(* CODESYS project codesys-poc

Project tree, tasks and I/O mapping:
  CODESYS_Control_RTE_V3 : CODESYS Control RTE V3, CODESYS, order no. 305017, version 3.5.21.10
    application Application
  Device : CODESYS Control Win V3 x64, CODESYS, version 3.5.21.10
    application Application
      libraries: Standard, 3.5.18.0 (System); Test Manager IEC Unit Test, 5.1.0.0 (Intern)
      task MainTask (cyclic, interval t#20ms, priority 1) calls PLC_PRG
      task VISU_TASK (cyclic, interval 100 ms, priority 31) calls VisuElems.Visu_Prg
      Antenna/
        function block Antenna [ST]: DiscesaAnteriore, DiscesaAnterioreEnabled, DiscesaAnterioreStop
        interface IAntenna: DiscesaAnteriore, DiscesaAnterioreEnabled, DiscesaAnterioreStop
        function block ManagerAntenna [ST]
      ArganoPrincipale/
        function block Argano [ST]: Arrotola
        interface IArgano: Arrotola
        function block ManagerArgano [ST]
      Controls/
        Joystyck/
          function block Joystick2 [CFC]
          function block Joystick3 [SFC]
          function block Joystick4 [FBD]
          function block Joystick [ST]
      Motore/
        interface IMotore: Accendi, GiriMotore, SpegniMotore
        function block MotoreDiesel [CFC]: Accendi, GiriMotore
      program PLC_PRG [ST]
      Rotary/
        interface IRotary: ClickClick, Rotate, RotateStop, SetCilindrata, SpinOff
        function block ManagerRotary [ST]
        function block Rotary [ST]: ClickClick, Rotate, RotateStop, SetCilindrata, SpinOff
        function block TestRotation_1 [ST]: Abort, Execute, Setup, Teardown
        function block TestRotation [ST]: Abort, Execute, Setup, Teardown
      Valvole/
        function block DistributoreValvole [ST]: openV1, openV2
        interface IDistributoreValvole: openV1, openV2
        interface IPompa: Portata
        function block Pompa [ST]: Portata
      visualisation Visualization_1
    application Application
      libraries: Standard, 3.5.18.0 (System)
      task MainTask (cyclic, interval t#20ms, priority 1) calls PLC_PRG
      task VISU_TASK (cyclic, interval 100 ms, priority 31) calls VisuElems.Visu_Prg
      Antenna/
        function block Antenna [ST]: DiscesaAnteriore, DiscesaAnterioreEnabled, DiscesaAnterioreStop
        interface IAntenna: DiscesaAnteriore, DiscesaAnterioreEnabled, DiscesaAnterioreStop
        function block ManagerAntenna [ST]
      ArganoPrincipale/
        function block Argano [ST]: Arrotola
        interface IArgano: Arrotola
        function block ManagerArgano [ST]
      Controls/
        Joystyck/
          function block Joystick2 [CFC]
          function block Joystick3 [SFC]
          function block Joystick4 [FBD]
          function block Joystick [ST]
      program PLC_PRG [ST]
      Rotary/
        interface IRotary: ClickClick, Rotate, RotateStop, SetCilindrata, SpinOff
        function block ManagerRotary [ST]
        function block Rotary [ST]: ClickClick, Rotate, RotateStop, SetCilindrata, SpinOff
      Valvole/
        function block DistributoreValvole [ST]: openV1, openV2
        interface IDistributoreValvole: openV1, openV2
        interface IPompa: Portata
        function block Pompa [ST]: Portata
      visualisation Visualization_1
    application Application
      libraries: Standard, 3.5.18.0 (System); Test Manager IEC Unit Test, 5.1.0.0 (Intern)
      task MainTask (cyclic, interval t#20ms, priority 1) calls PLC_PRG
      task VISU_TASK (cyclic, interval 100 ms, priority 31) calls VisuElems.Visu_Prg
      Antenna/
        function block Antenna [ST]: DiscesaAnteriore, DiscesaAnterioreEnabled, DiscesaAnterioreStop
        interface IAntenna: DiscesaAnteriore, DiscesaAnterioreEnabled, DiscesaAnterioreStop
        function block ManagerAntenna [ST]
      ArganoPrincipale/
        function block Argano [ST]: Arrotola
        interface IArgano: Arrotola
        function block ManagerArgano [ST]
      Controls/
        Joystyck/
          ClassDiagram_Control
          interface IJoystick: axisX, axisY, enabled, triggered
          function block Joystick2 [CFC]
          function block Joystick3 [SFC]
          function block Joystick4 [FBD]: axisX, axisY, enabled, safe, triggered
          function block Joystick [ST]: axisX, axisY, enabled, safe, triggered
      interface ISafeManaged: safe
      Motore/
        interface IMotore: Accendi, GiriMotore, SpegniMotore
        function block MotoreDiesel [CFC]: Accendi, GiriMotore
      program PLC_PRG [ST]
      Rotary/
        function block AutoRotate [CFC]: direction, enabled, speed
        ClassDiagram
        interface IAutoRotate: direction, enabled, speed
        interface IRotary: ClickClick, Rotate, RotateStop, SetCilindrata, SpinOff
        function block ManagerRotary [ST]
        function block Rotary [ST]: ClickClick, Rotate, RotateStop, safe, SetCilindrata, SpinOff
        function block TestRotation_1 [ST]: Abort, Execute, Setup, Teardown
        function block TestRotation [ST]: Abort, Execute, Setup, Teardown
      Valvole/
        function block DistributionValve [ST]: GetActual, GetTarget, Open, safe, openV2
        interface IDistributionValve: GetActual, GetTarget, Open, openV2
        interface IPompa: Portata
        function block Pompa [ST]: Portata
      visualisation Visualization_1
  Generated Unit Tests/
  text list GlobalTextList
*)

// Device/Application/PLC_PRG
PROGRAM PLC_PRG
VAR
	joystick1 : Joystick;
    joystick : Joystick4;
	
    rotary : Rotary;
	managerRotary: ManagerRotary;
	
	antenna: Antenna;
	managerAntenna: ManagerAntenna;
	
	argano: Argano;
	managerArgano: ManagerArgano;
	
	pompa : Pompa;
	distributore: DistributoreValvole;
	
	safe : BOOL;
	// Generated by IEC Unit Test
	xDone: BOOL;
	// Generated by IEC Unit Test
	xError: BOOL;
	// Generated by IEC Unit Test
	instTESTCASE: TestRotation;
END_VAR

joystick1.Safe := safe;
joystick.Safe := safe;

distributore.pompa := pompa;

managerRotary.joystick := joystick1;
managerRotary.rotary := rotary;

managerAntenna.joystick := joystick;
managerAntenna.antenna := antenna;

managerArgano.argano := argano;
managerArgano.antenna := antenna;

rotary.Safe := safe;
rotary.distributore := distributore;

// controlli
joystick();
joystick1();

// gruppi
antenna();
argano();
pompa();
distributore();

// manager
managerRotary();
managerAntenna(); // managerAntenna(antenna := antenna, joystick := joystick);
managerArgano();

END_PROGRAM

// Device/Application/Controls/Joystyck/Joystick
FUNCTION_BLOCK Joystick
VAR_INPUT
	Safe: BOOL;
	Trigger: BOOL;
END_VAR
VAR_OUTPUT
	Enabled: BOOL;
	EnabledOR: BOOL;
END_VAR
VAR
	EnabledInner: BOOL;
END_VAR

Enabled := Safe AND Trigger;
EnabledOR := Safe OR Trigger;

END_FUNCTION_BLOCK

// Device/Application/Controls/Joystyck/Joystick
FUNCTION_BLOCK Joystick
VAR_INPUT
	Safe: BOOL;
	Trigger: BOOL;
END_VAR
VAR_OUTPUT
	Enabled: BOOL;
	EnabledOR: BOOL;
END_VAR
VAR
	EnabledInner: BOOL;
END_VAR

Enabled := Safe AND Trigger;
EnabledOR := Safe OR Trigger;

END_FUNCTION_BLOCK

// Device/Application/Controls/Joystyck/Joystick
FUNCTION_BLOCK Joystick
VAR_INPUT
	Safe: BOOL;
	Trigger: BOOL;
END_VAR
VAR_OUTPUT
	Enabled: BOOL;
	EnabledOR: BOOL;
END_VAR
VAR
	EnabledInner: BOOL;
END_VAR

Enabled := Safe AND Trigger;
EnabledOR := Safe OR Trigger;

{warning 'Aggiungi implementazione della proprietà'}
PROPERTY axisX : REAL
GET
END_GET
END_PROPERTY

{warning 'Aggiungi implementazione della proprietà'}
PROPERTY axisY : REAL
GET
axisY := 0.0;
END_GET
END_PROPERTY

{warning 'Aggiungi implementazione della proprietà'}
PROPERTY enabled : BOOL
GET
END_GET
END_PROPERTY

{warning 'Aggiungi implementazione della proprietà'}
PROPERTY safe : BOOL
GET
safe := _safe;
END_GET
END_PROPERTY

{warning 'Aggiungi implementazione della proprietà'}
PROPERTY triggered : BOOL
GET
END_GET
END_PROPERTY

END_FUNCTION_BLOCK

// Device/Application/Valvole/Pompa
FUNCTION_BLOCK Pompa IMPLEMENTS IPompa
VAR_INPUT
	_portata: REAL;
END_VAR
VAR_OUTPUT
END_VAR
VAR
END_VAR

PROPERTY Portata : REAL
GET
Portata := _portata;
END_GET
SET
_portata := Portata;
END_SET
END_PROPERTY

END_FUNCTION_BLOCK

// Device/Application/Valvole/Pompa
FUNCTION_BLOCK Pompa IMPLEMENTS IPompa
VAR_INPUT
	_portata: REAL;
END_VAR
VAR_OUTPUT
END_VAR
VAR
END_VAR

PROPERTY Portata : REAL
GET
Portata := _portata;
END_GET
SET
_portata := Portata;
END_SET
END_PROPERTY

END_FUNCTION_BLOCK

// Device/Application/Valvole/Pompa
FUNCTION_BLOCK Pompa IMPLEMENTS IPompa
VAR_INPUT
	_portata: REAL;
END_VAR
VAR_OUTPUT
END_VAR
VAR
END_VAR

PROPERTY Portata : REAL
GET
Portata := _portata;
END_GET
SET
_portata := Portata;
END_SET
END_PROPERTY

END_FUNCTION_BLOCK

// Device/Application/Valvole/IPompa
INTERFACE IPompa

PROPERTY Portata : REAL
GET
END_GET
SET
END_SET
END_PROPERTY

END_INTERFACE

// Device/Application/Valvole/IPompa
INTERFACE IPompa

PROPERTY Portata : REAL
GET
END_GET
SET
END_SET
END_PROPERTY

END_INTERFACE

// Device/Application/Valvole/IPompa
INTERFACE IPompa

PROPERTY Portata : REAL
GET
END_GET
SET
END_SET
END_PROPERTY

END_INTERFACE

// Device/Application/Rotary/ManagerRotary
FUNCTION_BLOCK ManagerRotary
VAR_INPUT
	rotary: IRotary;
	joystick: Joystick;
END_VAR
VAR_OUTPUT
END_VAR
VAR
	rotationEnabled: BOOL;
END_VAR

// rotary.rotate = joystick.Enabled;
rotationEnabled := joystick.Enabled;

// SOL 1
IF rotationEnabled THEN
	rotary.Rotate(Side := 'LEFT', Speed := 10);
	// rampa(actual, desired);
ELSE
	rotary.RotateStop();
	// rotary.Rotate(Side := 'null', Speed := 0);
	// rampa(actual, 0);
END_IF

// SOL 2
//
// ManagerRotary:
//
// rotary.Rotate(rotationEnabled, Side := 'LEFT', Speed := 10);
//
// Rotary:
//
// IF rotationEnabled THEN
// 	  Rotate(rotationEnabled, Side := 'LEFT', Speed := 10);
// ELSE
// 	  Rotate(rotationEnabled, Side := 'LEFT', Speed := 0);
// END_IF


// SOL 3
//
// rotary.RotateStop(); SOLO SE FARE LO STOP E' IDEMPOTENTE
// IF rotationEnabled THEN
// 	rotary.Rotate(Side := 'LEFT', Speed := 10);
// END_IF

END_FUNCTION_BLOCK

// Device/Application/Rotary/Rotary
FUNCTION_BLOCK Rotary IMPLEMENTS IRotary
VAR_INPUT
	Safe: BOOL;
	distributore: IDistributoreValvole;
END_VAR
VAR_OUTPUT
END_VAR
VAR
    InvocationCount : INT := 0; // Counter for total method invocations
END_VAR

METHOD ClickClick
VAR
    clicked : BOOL;
END_VAR
// Simulate click-click behavior
clicked := TRUE; // Placeholder for actual logic

// IF Safe THEN
// 	InvocationCount := InvocationCount + 1; // Increase method call count
// END_IF;
END_METHOD

METHOD Rotate
VAR_INPUT
    Side : STRING;  // "Left" or "Right"
    Speed : REAL;   // Rotation speed
END_VAR
VAR_OUTPUT
	ActualSpeed: REAL;
END_VAR
// Simulated behavior
// direction := TO_UPPER(Side);
IF Side = 'LEFT' THEN
    // Do something for left rotation
    // For demo, just print or simulate log
    ; // Can add logging or effect
ELSIF Side = 'RIGHT' THEN
    // Do something for right rotation
    ;
ELSE
    ; // Invalid direction
END_IF;

InvocationCount := InvocationCount + 1; // Increase method call count
distributore.openV1(Speed);
ActualSpeed := Speed;
END_METHOD

METHOD RotateStop
distributore.openV1(0.0);
END_METHOD

METHOD SetCilindrata
// IF Safe THEN
// 	InvocationCount := InvocationCount + 1; // Increase method call count
// END_IF;
END_METHOD

METHOD SpinOff
VAR_INPUT
    dummy : BOOL;
END_VAR
// Simulate spinoff behavior
// For example: Do something when spinning off

// IF Safe THEN
// 	InvocationCount := InvocationCount + 1; // Increase method call count
// END_IF;
END_METHOD

END_FUNCTION_BLOCK

// Device/Application/Rotary/Rotary
FUNCTION_BLOCK Rotary IMPLEMENTS IRotary
VAR_INPUT
	Safe: BOOL;
	distributore: IDistributoreValvole;
END_VAR
VAR_OUTPUT
END_VAR
VAR
    InvocationCount : INT := 0; // Counter for total method invocations
END_VAR

METHOD ClickClick
VAR
    clicked : BOOL;
END_VAR
// Simulate click-click behavior
clicked := TRUE; // Placeholder for actual logic

// IF Safe THEN
// 	InvocationCount := InvocationCount + 1; // Increase method call count
// END_IF;
END_METHOD

METHOD Rotate
VAR_INPUT
    Side : STRING;  // "Left" or "Right"
    Speed : REAL;   // Rotation speed
END_VAR
VAR
    direction : STRING;
END_VAR
// Simulated behavior
// direction := TO_UPPER(Side);
IF Side = 'LEFT' THEN
    // Do something for left rotation
    // For demo, just print or simulate log
    ; // Can add logging or effect
ELSIF Side = 'RIGHT' THEN
    // Do something for right rotation
    ;
ELSE
    ; // Invalid direction
END_IF;

InvocationCount := InvocationCount + 1; // Increase method call count
distributore.openV1(10.0);
END_METHOD

METHOD RotateStop
distributore.openV1(0.0);
END_METHOD

METHOD SetCilindrata
// IF Safe THEN
// 	InvocationCount := InvocationCount + 1; // Increase method call count
// END_IF;
END_METHOD

METHOD SpinOff
VAR_INPUT
    dummy : BOOL;
END_VAR
// Simulate spinoff behavior
// For example: Do something when spinning off

// IF Safe THEN
// 	InvocationCount := InvocationCount + 1; // Increase method call count
// END_IF;
END_METHOD

END_FUNCTION_BLOCK

// Device/Application/Rotary/Rotary
FUNCTION_BLOCK Rotary IMPLEMENTS IRotary, ISafeManaged
VAR_INPUT
	distributore: IDistributionValve;
END_VAR
VAR_OUTPUT
END_VAR
VAR
    _safe: BOOL;
	invocationCount : INT := 0; // Counter for total method invocations
END_VAR

METHOD ClickClick
VAR
    clicked : BOOL;
END_VAR
// Simulate click-click behavior
clicked := TRUE; // Placeholder for actual logic

// IF Safe THEN
// 	InvocationCount := InvocationCount + 1; // Increase method call count
// END_IF;
END_METHOD

METHOD Rotate
VAR_INPUT
    side : STRING;  // "Left" or "Right"
    speed : REAL;   // Rotation speed
END_VAR
VAR_OUTPUT
	actualSpeed: REAL;
END_VAR
// Simulated behavior
// direction := TO_UPPER(Side);
IF Side = 'LEFT' THEN
    // Do something for left rotation
    // For demo, just print or simulate log
    ; // Can add logging or effect
ELSIF Side = 'RIGHT' THEN
    // Do something for right rotation
    ;
ELSE
    ; // Invalid direction
END_IF;

invocationCount := invocationCount + 1; // Increase method call count
distributionValve.Open(1, Speed);
actualSpeed := speed;
END_METHOD

METHOD RotateStop
distributionValve.open(1, 0.0);
END_METHOD

{warning 'Aggiungi implementazione della proprietà'}
PROPERTY safe : BOOL
GET
safe := _safe;
END_GET
END_PROPERTY

METHOD SetCilindrata
// IF Safe THEN
// 	InvocationCount := InvocationCount + 1; // Increase method call count
// END_IF;
END_METHOD

METHOD SpinOff
VAR_INPUT
    dummy : BOOL;
END_VAR
// Simulate spinoff behavior
// For example: Do something when spinning off

// IF Safe THEN
// 	InvocationCount := InvocationCount + 1; // Increase method call count
// END_IF;
END_METHOD

END_FUNCTION_BLOCK

// Device/Application/Rotary/IRotary
INTERFACE IRotary

METHOD ClickClick
VAR_INPUT
END_VAR
END_METHOD

METHOD Rotate
VAR_INPUT
    Side : STRING;  // "Left" or "Right"
    Speed : REAL;   // Rotation speed
END_VAR
VAR_OUTPUT
	ActualSpeed: REAL;
END_VAR
END_METHOD

METHOD RotateStop
VAR_INPUT
END_VAR
END_METHOD

METHOD SetCilindrata
VAR_INPUT
END_VAR
END_METHOD

METHOD SpinOff
VAR_INPUT
    dummy : BOOL;
END_VAR
END_METHOD

END_INTERFACE

// Device/Application/Rotary/IRotary
INTERFACE IRotary

METHOD ClickClick
VAR_INPUT
END_VAR
END_METHOD

METHOD Rotate
VAR_INPUT
    Side : STRING;  // "Left" or "Right"
    Speed : REAL;   // Rotation speed
END_VAR
END_METHOD

METHOD RotateStop
VAR_INPUT
END_VAR
END_METHOD

METHOD SetCilindrata
VAR_INPUT
END_VAR
END_METHOD

METHOD SpinOff
VAR_INPUT
    dummy : BOOL;
END_VAR
END_METHOD

END_INTERFACE

// Device/Application/Rotary/IRotary
INTERFACE IRotary

METHOD ClickClick
VAR_INPUT
END_VAR
END_METHOD

METHOD Rotate
VAR_INPUT
    Side : STRING;  // "Left" or "Right"
    Speed : REAL;   // Rotation speed
END_VAR
VAR_OUTPUT
	ActualSpeed: REAL;
END_VAR
END_METHOD

METHOD RotateStop
VAR_INPUT
END_VAR
END_METHOD

METHOD SetCilindrata
VAR_INPUT
END_VAR
END_METHOD

METHOD SpinOff
END_METHOD

END_INTERFACE

// Device/Application/ISafeManaged
INTERFACE ISafeManaged

PROPERTY safe : BOOL
GET
END_GET
END_PROPERTY

END_INTERFACE

// Device/Application/Valvole/IDistributionValve
INTERFACE IDistributionValve

METHOD GetActual : REAL
VAR_INPUT
	idValve: INT;
END_VAR
END_METHOD

METHOD GetTarget : REAL
VAR_INPUT
	idValve : INT;
END_VAR
END_METHOD

METHOD Open
VAR_INPUT
	idValve: INT;
	flow: REAL;
END_VAR
END_METHOD

METHOD openV2
VAR_INPUT
	portata: REAL;
END_VAR
END_METHOD

END_INTERFACE

// Device/Application/Valvole/DistributionValve
FUNCTION_BLOCK DistributionValve IMPLEMENTS IDistributionValve, ISafeManaged
VAR_INPUT
	pump : IPump;
END_VAR
VAR_OUTPUT
END_VAR
VAR
	_vActual: ARRAY[1..10] OF REAL := [0, 0, 0, 0, 0, 0, 0, 0, 0, 0];
	_vTarget: ARRAY[1..10] OF REAL := [0, 0, 0, 0, 0, 0, 0, 0, 0, 0];
	flowSum : REAL := 0.0; // Reset flow accumulator
	firstValve: INT := -1;
	i: INT := 1;
	count: INT := 0;
END_VAR

flowSum := 0.0; // Reset flow accumulator

FOR i := 1 TO 10 DO
    IF _vTarget[i] <> 0 THEN
		flowSum := flowSum + _vActual[i];        
		count := count + 1;
		_vActual[i] := _vTarget[i];
		firstValve := i;
    ELSE
        _vActual[i] := 0.0;
    END_IF
END_FOR

IF count = 1 THEN
	pump.flow := _vActual[firstValve];	
	_vActual[firstValve] := 100.0;
ELSE 
	pump.flow := flowSum;
END_IF

METHOD GetActual : REAL
VAR_INPUT
	idValve	: INT;
END_VAR
getActual := _vActual[idValve];
END_METHOD

METHOD GetTarget : REAL
VAR_INPUT
	idValve : INT;
END_VAR
getTarget := _vTarget[idValve];
END_METHOD

METHOD Open
VAR_INPUT
	idValve: INT;	
	flow: REAL;
END_VAR
_vTarget[idValve] := flow;
END_METHOD

{warning 'Aggiungi implementazione della proprietà'}
PROPERTY safe : BOOL
GET
END_GET
END_PROPERTY

METHOD openV2
VAR_INPUT
	portata: REAL;
END_VAR
_v2 := portata;
END_METHOD

END_FUNCTION_BLOCK

// Device/Application/Valvole/IDistributoreValvole
INTERFACE IDistributoreValvole

METHOD openV1
VAR_INPUT
	portata: REAL;
END_VAR
END_METHOD

METHOD openV2
VAR_INPUT
	portata: REAL;
END_VAR
END_METHOD

END_INTERFACE

// Device/Application/Valvole/IDistributoreValvole
INTERFACE IDistributoreValvole

METHOD openV1
VAR_INPUT
	portata: REAL;
END_VAR
END_METHOD

METHOD openV2
VAR_INPUT
	portata: REAL;
END_VAR
END_METHOD

END_INTERFACE

// Device/Application/Rotary/ManagerRotary
FUNCTION_BLOCK ManagerRotary
VAR_INPUT
	rotary: IRotary;
	joystick: Joystick;
END_VAR
VAR_OUTPUT
END_VAR
VAR
	rotationEnabled: BOOL;
END_VAR

// rotary.rotate = joystick.Enabled;
rotationEnabled := joystick.Enabled;

// SOL 1
IF rotationEnabled THEN
	rotary.Rotate(Side := 'LEFT', Speed := 10);
	// rampa(actual, desired);
ELSE
	// rotary.RotateStop();
	rotary.Rotate(Side := 'null', Speed := 0);
	// rampa(actual, 0);
END_IF

// SOL 2
//
// ManagerRotary:
//
// rotary.Rotate(rotationEnabled, Side := 'LEFT', Speed := 10);
//
// Rotary:
//
// IF rotationEnabled THEN
// 	  Rotate(rotationEnabled, Side := 'LEFT', Speed := 10);
// ELSE
// 	  Rotate(rotationEnabled, Side := 'LEFT', Speed := 0);
// END_IF


// SOL 3
//
// rotary.RotateStop(); SOLO SE FARE LO STOP E' IDEMPOTENTE
// IF rotationEnabled THEN
// 	rotary.Rotate(Side := 'LEFT', Speed := 10);
// END_IF

END_FUNCTION_BLOCK

// Device/Application/Rotary/ManagerRotary
FUNCTION_BLOCK ManagerRotary
VAR_INPUT
	rotary: IRotary;
	joystick: IJoystick;
END_VAR
VAR_OUTPUT
END_VAR
VAR
	_rotationEnabled: BOOL;
END_VAR

// rotary.rotate = joystick.Enabled;
_rotationEnabled := joystick.Enabled;

// SOL 1
IF _rotationEnabled THEN
	rotary.Rotate(Side := 'LEFT', Speed := 10);
	// rampa(actual, desired);
ELSE
	rotary.RotateStop();
	// rotary.Rotate(Side := 'null', Speed := 0);
	// rampa(actual, 0);
END_IF

// SOL 2
//
// ManagerRotary:
//
// rotary.Rotate(rotationEnabled, Side := 'LEFT', Speed := 10);
//
// Rotary:
//
// IF rotationEnabled THEN
// 	  Rotate(rotationEnabled, Side := 'LEFT', Speed := 10);
// ELSE
// 	  Rotate(rotationEnabled, Side := 'LEFT', Speed := 0);
// END_IF


// SOL 3
//
// rotary.RotateStop(); SOLO SE FARE LO STOP E' IDEMPOTENTE
// IF rotationEnabled THEN
// 	rotary.Rotate(Side := 'LEFT', Speed := 10);
// END_IF

END_FUNCTION_BLOCK

// Device/Application/Controls/Joystyck/IJoystick
INTERFACE IJoystick EXTENDS ISafeManaged

PROPERTY axisX : REAL
GET
END_GET
END_PROPERTY

PROPERTY axisY : REAL
GET
END_GET
END_PROPERTY

PROPERTY enabled : BOOL
GET
END_GET
END_PROPERTY

PROPERTY triggered : BOOL
GET
END_GET
END_PROPERTY

END_INTERFACE

// Device/Application/Antenna/ManagerAntenna
FUNCTION_BLOCK ManagerAntenna
VAR_INPUT
	antenna: IAntenna;
	joystick: Joystick4;
END_VAR
VAR_OUTPUT
END_VAR
VAR
END_VAR

IF joystick.Enabled THEN
	antenna.DiscesaAnteriore();
ELSE
	antenna.DiscesaAnterioreStop();
END_IF

END_FUNCTION_BLOCK

// Device/Application/Antenna/Antenna
FUNCTION_BLOCK Antenna IMPLEMENTS IAntenna
VAR
	_discesaanterioreenabled : BOOL := FALSE; // Internal state
END_VAR

METHOD DiscesaAnteriore
_discesaanterioreenabled := TRUE;
END_METHOD

PROPERTY PUBLIC DiscesaAnterioreEnabled : BOOL
GET
DiscesaAnterioreEnabled := _discesaanterioreenabled;
END_GET
END_PROPERTY

METHOD DiscesaAnterioreStop
_discesaanterioreenabled := FALSE;
END_METHOD

END_FUNCTION_BLOCK

// Device/Application/Antenna/Antenna
FUNCTION_BLOCK Antenna IMPLEMENTS IAntenna
VAR
	_discesaanterioreenabled : BOOL := FALSE; // Internal state
END_VAR

METHOD DiscesaAnteriore
_discesaanterioreenabled := TRUE;
END_METHOD

PROPERTY PUBLIC DiscesaAnterioreEnabled : BOOL
GET
DiscesaAnterioreEnabled := _discesaanterioreenabled;
END_GET
END_PROPERTY

METHOD DiscesaAnterioreStop
_discesaanterioreenabled := FALSE;
END_METHOD

END_FUNCTION_BLOCK

// Device/Application/Antenna/Antenna
FUNCTION_BLOCK Antenna IMPLEMENTS IAntenna
VAR
	_discesaanterioreenabled : BOOL := FALSE; // Internal state
END_VAR

METHOD DiscesaAnteriore
_discesaanterioreenabled := TRUE;
END_METHOD

PROPERTY PUBLIC DiscesaAnterioreEnabled : BOOL
GET
DiscesaAnterioreEnabled := _discesaanterioreenabled;
END_GET
END_PROPERTY

METHOD DiscesaAnterioreStop
_discesaanterioreenabled := FALSE;
END_METHOD

END_FUNCTION_BLOCK

// Device/Application/Antenna/IAntenna
INTERFACE IAntenna

METHOD DiscesaAnteriore
VAR_INPUT
END_VAR
END_METHOD

PROPERTY PUBLIC DiscesaAnterioreEnabled : BOOL
GET
END_GET
END_PROPERTY

METHOD DiscesaAnterioreStop
VAR_INPUT
END_VAR
END_METHOD

END_INTERFACE

// Device/Application/Antenna/IAntenna
INTERFACE IAntenna

METHOD DiscesaAnteriore
VAR_INPUT
END_VAR
END_METHOD

PROPERTY PUBLIC DiscesaAnterioreEnabled : BOOL
GET
END_GET
END_PROPERTY

METHOD DiscesaAnterioreStop
VAR_INPUT
END_VAR
END_METHOD

END_INTERFACE

// Device/Application/Antenna/IAntenna
INTERFACE IAntenna

METHOD DiscesaAnteriore
VAR_INPUT
END_VAR
END_METHOD

PROPERTY PUBLIC DiscesaAnterioreEnabled : BOOL
GET
END_GET
END_PROPERTY

METHOD DiscesaAnterioreStop
VAR_INPUT
END_VAR
END_METHOD

END_INTERFACE

// Device/Application/Antenna/ManagerAntenna
FUNCTION_BLOCK ManagerAntenna
VAR_INPUT
	antenna: IAntenna;
	joystick: Joystick4;
END_VAR
VAR_OUTPUT
END_VAR
VAR
END_VAR

IF joystick.Enabled THEN
	antenna.DiscesaAnteriore();
ELSE
	antenna.DiscesaAnterioreStop();
END_IF

END_FUNCTION_BLOCK

// Device/Application/Antenna/ManagerAntenna
FUNCTION_BLOCK ManagerAntenna
VAR_INPUT
	antenna: IAntenna;
	joystick: Joystick4;
END_VAR
VAR_OUTPUT
END_VAR
VAR
END_VAR

IF joystick.Enabled THEN
	antenna.DiscesaAnteriore();
ELSE
	antenna.DiscesaAnterioreStop();
END_IF

END_FUNCTION_BLOCK

// Device/Application/Controls/Joystyck/Joystick4
FUNCTION_BLOCK Joystick4
VAR_INPUT
	Safe: BOOL;
END_VAR
VAR_OUTPUT
	Enabled: BOOL;
END_VAR
VAR
	Trigger: BOOL;
END_VAR

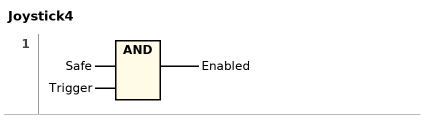
// NETWORK 1
Enabled := Safe AND Trigger;

END_FUNCTION_BLOCK

// Device/Application/Controls/Joystyck/Joystick4
FUNCTION_BLOCK Joystick4
VAR_INPUT
	Safe: BOOL;
END_VAR
VAR_OUTPUT
	Enabled: BOOL;
END_VAR
VAR
	Trigger: BOOL;
END_VAR

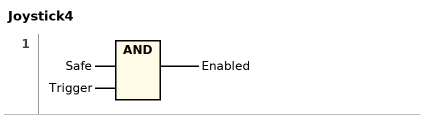
// NETWORK 1
Enabled := Safe AND Trigger;

END_FUNCTION_BLOCK

// Device/Application/Controls/Joystyck/Joystick4
FUNCTION_BLOCK Joystick4
VAR_INPUT
	Safe: BOOL;
END_VAR
VAR_OUTPUT
	Enabled: BOOL;
END_VAR
VAR
	Trigger: BOOL;
END_VAR

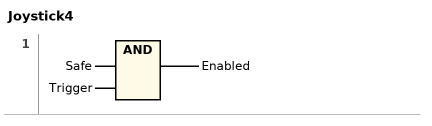
// NETWORK 1
Enabled := Safe AND Trigger;

{warning 'Aggiungi implementazione della proprietà'}
PROPERTY axisX : REAL
GET
END_GET
END_PROPERTY

{warning 'Aggiungi implementazione della proprietà'}
PROPERTY axisY : REAL
GET
END_GET
END_PROPERTY

{warning 'Aggiungi implementazione della proprietà'}
PROPERTY enabled : BOOL
GET
END_GET
END_PROPERTY

{warning 'Aggiungi implementazione della proprietà'}
PROPERTY safe : BOOL
GET
END_GET
END_PROPERTY

{warning 'Aggiungi implementazione della proprietà'}
PROPERTY triggered : BOOL
GET
END_GET
END_PROPERTY

END_FUNCTION_BLOCK

// Device/Application/ArganoPrincipale/ManagerArgano
FUNCTION_BLOCK ManagerArgano
VAR_INPUT
	argano: IArgano;
	antenna: IAntenna;
END_VAR
VAR_OUTPUT
END_VAR
VAR
	foo : BOOL := TRUE;
END_VAR

IF antenna.DiscesaAnterioreEnabled THEN
	argano.Arrotola();
END_IF

foo := not foo;

END_FUNCTION_BLOCK

// Device/Application/ArganoPrincipale/Argano
FUNCTION_BLOCK Argano IMPLEMENTS IArgano
VAR_INPUT
END_VAR
VAR_OUTPUT
END_VAR
VAR
	foo : BOOL := FALSE;
END_VAR

METHOD Arrotola
foo := not foo;
END_METHOD

END_FUNCTION_BLOCK

// Device/Application/ArganoPrincipale/Argano
FUNCTION_BLOCK Argano IMPLEMENTS IArgano
VAR_INPUT
END_VAR
VAR_OUTPUT
END_VAR
VAR
	foo : BOOL := FALSE;
END_VAR

METHOD Arrotola
foo := not foo;
END_METHOD

END_FUNCTION_BLOCK

// Device/Application/ArganoPrincipale/Argano
FUNCTION_BLOCK Argano IMPLEMENTS IArgano
VAR_INPUT
END_VAR
VAR_OUTPUT
END_VAR
VAR
	foo : BOOL := FALSE;
END_VAR

METHOD Arrotola
foo := not foo;
END_METHOD

END_FUNCTION_BLOCK

// Device/Application/ArganoPrincipale/IArgano
INTERFACE IArgano

METHOD Arrotola
VAR_INPUT
END_VAR
END_METHOD

END_INTERFACE

// Device/Application/ArganoPrincipale/IArgano
INTERFACE IArgano

METHOD Arrotola
VAR_INPUT
END_VAR
END_METHOD

END_INTERFACE

// Device/Application/ArganoPrincipale/IArgano
INTERFACE IArgano

METHOD Arrotola
VAR_INPUT
END_VAR
END_METHOD

END_INTERFACE

// Device/Application/ArganoPrincipale/ManagerArgano
FUNCTION_BLOCK ManagerArgano
VAR_INPUT
	argano: IArgano;
	antenna: IAntenna;
END_VAR
VAR_OUTPUT
END_VAR
VAR
	foo : BOOL := TRUE;
END_VAR

IF antenna.DiscesaAnterioreEnabled THEN
	argano.Arrotola();
END_IF

foo := not foo;

END_FUNCTION_BLOCK

// Device/Application/ArganoPrincipale/ManagerArgano
FUNCTION_BLOCK ManagerArgano
VAR_INPUT
	argano: IArgano;
	antenna: IAntenna;
END_VAR
VAR_OUTPUT
END_VAR
VAR
	foo : BOOL := TRUE;
END_VAR

IF antenna.DiscesaAnterioreEnabled THEN
	argano.Arrotola();
END_IF

foo := not foo;

END_FUNCTION_BLOCK

// Device/Application/PLC_PRG
PROGRAM PLC_PRG
VAR
	joystick1 : Joystick;
    joystick : Joystick4;
	
    rotary : Rotary;
	managerRotary: ManagerRotary;
	
	antenna: Antenna;
	managerAntenna: ManagerAntenna;
	
	argano: Argano;
	managerArgano: ManagerArgano;
	
	pompa : Pompa;
	distributore: DistributoreValvole;
	
	safe : BOOL;
END_VAR

joystick1.Safe := safe;
joystick.Safe := safe;

distributore.pompa := pompa;

managerRotary.joystick := joystick1;
managerRotary.rotary := rotary;

managerAntenna.joystick := joystick;
managerAntenna.antenna := antenna;

managerArgano.argano := argano;
managerArgano.antenna := antenna;

rotary.Safe := Safe;
rotary.distributore := distributore;

// controlli
joystick();
joystick1();

// gruppi
antenna();
argano();
pompa();
distributore();

// manager
managerRotary();
managerAntenna(); // managerAntenna(antenna := antenna, joystick := joystick);
managerArgano();

END_PROGRAM

// Device/Application/PLC_PRG
PROGRAM PLC_PRG
VAR
	joystick : Joystick;
	
    rotary : Rotary;
	managerRotary: ManagerRotary;
	
	antenna: Antenna;
	managerAntenna: ManagerAntenna;
	
	argano: Argano;
	managerArgano: ManagerArgano;
	
	pompa : Pump;
	distributore: DistributionValve;
	
	safe : BOOL;
END_VAR

// lettura della parte SAFE

// configurazione

joystick.safe := safe;

distributore.pump := pompa;

managerRotary.joystick := joystick;
managerRotary.rotary := rotary;

managerAntenna.joystick := joystick;
managerAntenna.antenna := antenna;

managerArgano.argano := argano;
managerArgano.antenna := antenna;

// controlli
joystick();

// gruppi
rotary(_safe := safe, _distributore := distributore);
antenna();
argano();
pompa();
distributore();

// manager
managerRotary();
managerAntenna(); // managerAntenna(antenna := antenna, joystick := joystick);
managerArgano();

END_PROGRAM

// Device/Application/Valvole/DistributoreValvole
FUNCTION_BLOCK DistributoreValvole IMPLEMENTS IDistributoreValvole
VAR_INPUT
	pompa : IPompa;
END_VAR
VAR_OUTPUT
END_VAR
VAR
	_v1: REAL;
	_v2: REAL;
	v1: REAL;
	v2: REAL;
	foo: BOOL := false;
END_VAR

v1 := _v1;
v2 := _v2;
IF _v1 = 0 AND _v2 <> 0 THEN
	v2 := 100.0;
	pompa.portata := _v2;
ELSIF _v2 = 0 AND _v1 <> 0 THEN
	v1 := 100.0;
	pompa.portata := _v1;
ELSIF _v2 <> 0 AND _v1 <> 0 THEN
	pompa.portata := v1 + v2;
ELSE
	pompa.portata := 0;
END_IF

METHOD openV1
VAR_INPUT
	portata: REAL;
END_VAR
_v1 := portata;
foo := not foo;
END_METHOD

METHOD openV2
VAR_INPUT
	portata: REAL;
END_VAR
_v2 := portata;
END_METHOD

END_FUNCTION_BLOCK

// Device/Application/Valvole/DistributoreValvole
FUNCTION_BLOCK DistributoreValvole IMPLEMENTS IDistributoreValvole
VAR_INPUT
	pompa : IPompa;
END_VAR
VAR_OUTPUT
END_VAR
VAR
	_v1: REAL;
	_v2: REAL;
	v1: REAL;
	v2: REAL;
	foo: BOOL := false;
END_VAR

v1 := _v1;
v2 := _v2;
IF _v1 = 0 AND _v2 <> 0 THEN
	v2 := 100.0;
	pompa.portata := _v2;
ELSIF _v2 = 0 AND _v1 <> 0 THEN
	v1 := 100.0;
	pompa.portata := _v1;
ELSIF _v2 <> 0 AND _v1 <> 0 THEN
	pompa.portata := v1 + v2;
ELSE
	pompa.portata := 0;
END_IF

METHOD openV1
VAR_INPUT
	portata: REAL;
END_VAR
_v1 := portata;
foo := not foo;
END_METHOD

METHOD openV2
VAR_INPUT
	portata: REAL;
END_VAR
_v2 := portata;
END_METHOD

END_FUNCTION_BLOCK

// Device/Application/Rotary/TestRotation
(*
    This is the recommended way to implement a single test case.
 
    The template ``TM.Testcase`` provides an easy to use pattern for a single test case.
    It consists of a set of methods and outputs to carry out test specific tasks. When the test is
    run, the POU's methods will be called in the following sequence:
    - ``Setup()`` (optional, called once) offers the possiblity to prepare testee and test.
    - ``Execute()`` (mandatory, called in the loop) is designed to stimulate the testee and check it's results. The method
      gets called, until it returns  ``TRUE``. The methods's VAR_OUTPUT ``iErrorCode`` is used to report
      success (0) or failure (<>0). The POU's VAR_OUTPUT ``sInfo`` is used to include textual details in the test report.
    - ``Teardown()`` (optional, called once) offers the possibility to clean up testee and reset the test after it
      finished.
     
    As the template implements the behaviour ``CBM.ETrigA``, it can be aborted. In that case the method
    ``Abort()`` will be called repeatedly, until it returns TRUE. This offers the possibility to clean up
    a running test in any state.
*)
{attribute 'test'}
{attribute 'testcasename':='TestRotazione'}
{attribute 'testcategory':='TestRotary'}
{attribute 'testcasetimeout':='15000'}
FUNCTION_BLOCK TestRotation EXTENDS TM.Testcase
VAR_INPUT
END_VAR
VAR_OUTPUT
END_VAR
VAR
	rotary: Rotary;
	distributore: DistributoreValvole;
END_VAR

SUPER^();   // mandatory - don't change

(*
    Overwrite this method, to perform cleanup actions when the test is to be aborted
    and return ``TRUE``, once you are finished.
     
    ``Abort()`` gets called to abort the current test. It is called repeatedly until it
    returns ``TRUE``.
     
    **DO NOT CALL** the base implementation ``SUPER^.Abort``, as this will simply return ``TRUE``.
     
    :return: ``FALSE`` - abort not finished, ```TRUE`` - abort finished
 *)
METHOD PROTECTED Abort : BOOL
// TODO Abort and clean up the running testee and test
 
Abort := TRUE;  // mandatory: signal abort completed
END_METHOD

(*
    Implement the logic of the testcase in this method.
 
    Once the test has been started, this method will be called until
    a) the method returns ``TRUE``, which signals completion of the test,
        or
    b) the test is aborted.
 
    Once this method returns ``TRUE``, the output iErrorCode is evaluated: The value 0
    signals success, while all other values signal a failure of the test.
    To provide additional information about the test, set the global output sInfo
    of the base FB.
         
    **DO NOT CALL** the base implementation of this method ``SUPER^.Execute()``.
     
    :return: ``FALSE`` - execution is not finished, ```TRUE`` - execution is finished
*)
METHOD PROTECTED Execute : BOOL
VAR_OUTPUT
	iErrorCode	: INT;
END_VAR
VAR
	ActualSpeed : REAL;
END_VAR

ActualSpeed := rotary.Rotate(Side := 'LEFT', Speed:= 10.0);
TM.Assert_Bool_IsTrue(context := THIS^, actualValue := ActualSpeed = 10.0, wsErrorMsg := "Dummy test result - change the test implementation.");
Execute := TRUE;
END_METHOD

(*
    Overwrite this method, if any preparations need done before the first call to ``Execute()``.   
    This optional method ``Setup()`` is called once before the test is started.
     
    The return value is ignored. Its sole purpose is to satisfy the compiler.
     
    When overwritten, it is **NOT REQUIRED** to call the base implementation ``SUPER^.Setup()``,
    as the base implementation is empty.
 *)
METHOD PROTECTED Setup : BOOL
rotary.Safe := TRUE;
rotary.distributore := distributore;
END_METHOD

(*
    Overwrite this method, to implement necessary teardown actions
    after the test is finished. For example reset additional outputs defined
    by your implementation.
     
    ``Teardown()`` is called once after the test is reset.
     
    The return value is ignored. Its sole purpose is to satisfy the compiler.
     
    When overwritten, it is **NOT REQUIRED** to call the base implementation ``SUPER^.Teardown()``,
    as the base implementation is empty.   
 *)
METHOD PROTECTED Teardown : BOOL
// TODO Clean up testee and test after test case finished
END_METHOD

END_FUNCTION_BLOCK

// Device/Application/Rotary/TestRotation
(*
    This is the recommended way to implement a single test case.
 
    The template ``TM.Testcase`` provides an easy to use pattern for a single test case.
    It consists of a set of methods and outputs to carry out test specific tasks. When the test is
    run, the POU's methods will be called in the following sequence:
    - ``Setup()`` (optional, called once) offers the possiblity to prepare testee and test.
    - ``Execute()`` (mandatory, called in the loop) is designed to stimulate the testee and check it's results. The method
      gets called, until it returns  ``TRUE``. The methods's VAR_OUTPUT ``iErrorCode`` is used to report
      success (0) or failure (<>0). The POU's VAR_OUTPUT ``sInfo`` is used to include textual details in the test report.
    - ``Teardown()`` (optional, called once) offers the possibility to clean up testee and reset the test after it
      finished.
     
    As the template implements the behaviour ``CBM.ETrigA``, it can be aborted. In that case the method
    ``Abort()`` will be called repeatedly, until it returns TRUE. This offers the possibility to clean up
    a running test in any state.
*)
{attribute 'test'}
{attribute 'testcasename':='TestRotazione'}
{attribute 'testcategory':='TestRotary'}
{attribute 'testcasetimeout':='15000'}
FUNCTION_BLOCK TestRotation EXTENDS TM.Testcase
VAR_INPUT
END_VAR
VAR_OUTPUT
END_VAR
VAR
	rotary: Rotary;
	distributore: DistributionValve;
END_VAR

SUPER^();   // mandatory - don't change

(*
    Overwrite this method, to perform cleanup actions when the test is to be aborted
    and return ``TRUE``, once you are finished.
     
    ``Abort()`` gets called to abort the current test. It is called repeatedly until it
    returns ``TRUE``.
     
    **DO NOT CALL** the base implementation ``SUPER^.Abort``, as this will simply return ``TRUE``.
     
    :return: ``FALSE`` - abort not finished, ```TRUE`` - abort finished
 *)
METHOD PROTECTED Abort : BOOL
// TODO Abort and clean up the running testee and test
 
Abort := TRUE;  // mandatory: signal abort completed
END_METHOD

(*
    Implement the logic of the testcase in this method.
 
    Once the test has been started, this method will be called until
    a) the method returns ``TRUE``, which signals completion of the test,
        or
    b) the test is aborted.
 
    Once this method returns ``TRUE``, the output iErrorCode is evaluated: The value 0
    signals success, while all other values signal a failure of the test.
    To provide additional information about the test, set the global output sInfo
    of the base FB.
         
    **DO NOT CALL** the base implementation of this method ``SUPER^.Execute()``.
     
    :return: ``FALSE`` - execution is not finished, ```TRUE`` - execution is finished
*)
METHOD PROTECTED Execute : BOOL
VAR_OUTPUT
	iErrorCode	: INT;
END_VAR
VAR
	ActualSpeed : REAL;
END_VAR

ActualSpeed := rotary.Rotate(Side := 'LEFT', Speed:= 10.0);
TM.Assert_Bool_IsTrue(context := THIS^, actualValue := ActualSpeed = 10.0, wsErrorMsg := "Dummy test result - change the test implementation.");
Execute := TRUE;
END_METHOD

(*
    Overwrite this method, if any preparations need done before the first call to ``Execute()``.   
    This optional method ``Setup()`` is called once before the test is started.
     
    The return value is ignored. Its sole purpose is to satisfy the compiler.
     
    When overwritten, it is **NOT REQUIRED** to call the base implementation ``SUPER^.Setup()``,
    as the base implementation is empty.
 *)
METHOD PROTECTED Setup : BOOL
rotary.Safe := TRUE;
rotary.distributionValve := distributore;
END_METHOD

(*
    Overwrite this method, to implement necessary teardown actions
    after the test is finished. For example reset additional outputs defined
    by your implementation.
     
    ``Teardown()`` is called once after the test is reset.
     
    The return value is ignored. Its sole purpose is to satisfy the compiler.
     
    When overwritten, it is **NOT REQUIRED** to call the base implementation ``SUPER^.Teardown()``,
    as the base implementation is empty.   
 *)
METHOD PROTECTED Teardown : BOOL
// TODO Clean up testee and test after test case finished
END_METHOD

END_FUNCTION_BLOCK

// Device/Application/Motore/IMotore
INTERFACE IMotore

METHOD Accendi
VAR_INPUT
END_VAR
END_METHOD

PROPERTY GiriMotore : INT
GET
END_GET
SET
END_SET
END_PROPERTY

METHOD SpegniMotore
VAR_INPUT
END_VAR
END_METHOD

END_INTERFACE

// Device/Application/Motore/IMotore
INTERFACE IMotore

METHOD Accendi
VAR_INPUT
END_VAR
END_METHOD

PROPERTY GiriMotore : INT
GET
END_GET
SET
END_SET
END_PROPERTY

METHOD SpegniMotore
VAR_INPUT
END_VAR
END_METHOD

END_INTERFACE

// Device/Application/Motore/MotoreDiesel
FUNCTION_BLOCK MotoreDiesel IMPLEMENTS IMotore
VAR_INPUT
END_VAR
VAR_OUTPUT
END_VAR
VAR
END_VAR


{warning 'Aggiungi implementazione del metodo'}
METHOD Accendi
END_METHOD

{warning 'Aggiungi implementazione della proprietà'}
PROPERTY GiriMotore : INT
GET
END_GET
SET
END_SET
END_PROPERTY

END_FUNCTION_BLOCK

// Device/Application/Motore/MotoreDiesel
FUNCTION_BLOCK MotoreDiesel IMPLEMENTS IMotore
VAR_INPUT
END_VAR
VAR_OUTPUT
END_VAR
VAR
END_VAR


{warning 'Aggiungi implementazione del metodo'}
METHOD Accendi
END_METHOD

{warning 'Aggiungi implementazione della proprietà'}
PROPERTY GiriMotore : INT
GET
END_GET
SET
END_SET
END_PROPERTY

END_FUNCTION_BLOCK

// Device/Application/Rotary/TestRotation_1
(*
    This is the recommended way to implement a single test case.
 
    The template ``TM.Testcase`` provides an easy to use pattern for a single test case.
    It consists of a set of methods and outputs to carry out test specific tasks. When the test is
    run, the POU's methods will be called in the following sequence:
    - ``Setup()`` (optional, called once) offers the possiblity to prepare testee and test.
    - ``Execute()`` (mandatory, called in the loop) is designed to stimulate the testee and check it's results. The method
      gets called, until it returns  ``TRUE``. The methods's VAR_OUTPUT ``iErrorCode`` is used to report
      success (0) or failure (<>0). The POU's VAR_OUTPUT ``sInfo`` is used to include textual details in the test report.
    - ``Teardown()`` (optional, called once) offers the possibility to clean up testee and reset the test after it
      finished.
     
    As the template implements the behaviour ``CBM.ETrigA``, it can be aborted. In that case the method
    ``Abort()`` will be called repeatedly, until it returns TRUE. This offers the possibility to clean up
    a running test in any state.
*)
{attribute 'test'}
{attribute 'testcasename':='TestRotazione'}
{attribute 'testcategory':='TestRotary'}
{attribute 'testcasetimeout':='15000'}
FUNCTION_BLOCK TestRotation_1 EXTENDS TM.Testcase
VAR_INPUT
END_VAR
VAR_OUTPUT
END_VAR
VAR
	rotary: Rotary;
	distributore: DistributoreValvole;
END_VAR

SUPER^();   // mandatory - don't change

(*
    Overwrite this method, to perform cleanup actions when the test is to be aborted
    and return ``TRUE``, once you are finished.
     
    ``Abort()`` gets called to abort the current test. It is called repeatedly until it
    returns ``TRUE``.
     
    **DO NOT CALL** the base implementation ``SUPER^.Abort``, as this will simply return ``TRUE``.
     
    :return: ``FALSE`` - abort not finished, ```TRUE`` - abort finished
 *)
METHOD PROTECTED Abort : BOOL
// TODO Abort and clean up the running testee and test
 
Abort := TRUE;  // mandatory: signal abort completed
END_METHOD

(*
    Implement the logic of the testcase in this method.
 
    Once the test has been started, this method will be called until
    a) the method returns ``TRUE``, which signals completion of the test,
        or
    b) the test is aborted.
 
    Once this method returns ``TRUE``, the output iErrorCode is evaluated: The value 0
    signals success, while all other values signal a failure of the test.
    To provide additional information about the test, set the global output sInfo
    of the base FB.
         
    **DO NOT CALL** the base implementation of this method ``SUPER^.Execute()``.
     
    :return: ``FALSE`` - execution is not finished, ```TRUE`` - execution is finished
*)
METHOD PROTECTED Execute : BOOL
VAR_OUTPUT
	iErrorCode	: INT;
END_VAR
VAR
	ActualSpeed : REAL;
END_VAR

ActualSpeed := rotary.Rotate(Side := 'LEFT', Speed:= 10.0);
TM.Assert_Bool_IsTrue(context := THIS^, actualValue := ActualSpeed = 10.0, wsErrorMsg := "Dummy test result - change the test implementation.");
Execute := TRUE;
END_METHOD

(*
    Overwrite this method, if any preparations need done before the first call to ``Execute()``.   
    This optional method ``Setup()`` is called once before the test is started.
     
    The return value is ignored. Its sole purpose is to satisfy the compiler.
     
    When overwritten, it is **NOT REQUIRED** to call the base implementation ``SUPER^.Setup()``,
    as the base implementation is empty.
 *)
METHOD PROTECTED Setup : BOOL
rotary.Safe := TRUE;
rotary.distributore := distributore;
END_METHOD

(*
    Overwrite this method, to implement necessary teardown actions
    after the test is finished. For example reset additional outputs defined
    by your implementation.
     
    ``Teardown()`` is called once after the test is reset.
     
    The return value is ignored. Its sole purpose is to satisfy the compiler.
     
    When overwritten, it is **NOT REQUIRED** to call the base implementation ``SUPER^.Teardown()``,
    as the base implementation is empty.   
 *)
METHOD PROTECTED Teardown : BOOL
// TODO Clean up testee and test after test case finished
END_METHOD

END_FUNCTION_BLOCK

// Device/Application/Rotary/TestRotation_1
(*
    This is the recommended way to implement a single test case.
 
    The template ``TM.Testcase`` provides an easy to use pattern for a single test case.
    It consists of a set of methods and outputs to carry out test specific tasks. When the test is
    run, the POU's methods will be called in the following sequence:
    - ``Setup()`` (optional, called once) offers the possiblity to prepare testee and test.
    - ``Execute()`` (mandatory, called in the loop) is designed to stimulate the testee and check it's results. The method
      gets called, until it returns  ``TRUE``. The methods's VAR_OUTPUT ``iErrorCode`` is used to report
      success (0) or failure (<>0). The POU's VAR_OUTPUT ``sInfo`` is used to include textual details in the test report.
    - ``Teardown()`` (optional, called once) offers the possibility to clean up testee and reset the test after it
      finished.
     
    As the template implements the behaviour ``CBM.ETrigA``, it can be aborted. In that case the method
    ``Abort()`` will be called repeatedly, until it returns TRUE. This offers the possibility to clean up
    a running test in any state.
*)
{attribute 'test'}
{attribute 'testcasename':='TestRotazione'}
{attribute 'testcategory':='TestRotary'}
{attribute 'testcasetimeout':='15000'}
FUNCTION_BLOCK TestRotation_1 EXTENDS TM.Testcase
VAR_INPUT
END_VAR
VAR_OUTPUT
END_VAR
VAR
	rotary: Rotary;
	distributore: DistributionValve;
END_VAR

SUPER^();   // mandatory - don't change

(*
    Overwrite this method, to perform cleanup actions when the test is to be aborted
    and return ``TRUE``, once you are finished.
     
    ``Abort()`` gets called to abort the current test. It is called repeatedly until it
    returns ``TRUE``.
     
    **DO NOT CALL** the base implementation ``SUPER^.Abort``, as this will simply return ``TRUE``.
     
    :return: ``FALSE`` - abort not finished, ```TRUE`` - abort finished
 *)
METHOD PROTECTED Abort : BOOL
// TODO Abort and clean up the running testee and test
 
Abort := TRUE;  // mandatory: signal abort completed
END_METHOD

(*
    Implement the logic of the testcase in this method.
 
    Once the test has been started, this method will be called until
    a) the method returns ``TRUE``, which signals completion of the test,
        or
    b) the test is aborted.
 
    Once this method returns ``TRUE``, the output iErrorCode is evaluated: The value 0
    signals success, while all other values signal a failure of the test.
    To provide additional information about the test, set the global output sInfo
    of the base FB.
         
    **DO NOT CALL** the base implementation of this method ``SUPER^.Execute()``.
     
    :return: ``FALSE`` - execution is not finished, ```TRUE`` - execution is finished
*)
METHOD PROTECTED Execute : BOOL
VAR_OUTPUT
	iErrorCode	: INT;
END_VAR
VAR
	ActualSpeed : REAL;
END_VAR

ActualSpeed := rotary.Rotate(Side := 'LEFT', Speed:= 10.0);
TM.Assert_Bool_IsTrue(context := THIS^, actualValue := ActualSpeed = 10.0, wsErrorMsg := "Dummy test result - change the test implementation.");
Execute := TRUE;
END_METHOD

(*
    Overwrite this method, if any preparations need done before the first call to ``Execute()``.   
    This optional method ``Setup()`` is called once before the test is started.
     
    The return value is ignored. Its sole purpose is to satisfy the compiler.
     
    When overwritten, it is **NOT REQUIRED** to call the base implementation ``SUPER^.Setup()``,
    as the base implementation is empty.
 *)
METHOD PROTECTED Setup : BOOL
rotary.Safe := TRUE;
rotary.distributore := distributore;
END_METHOD

(*
    Overwrite this method, to implement necessary teardown actions
    after the test is finished. For example reset additional outputs defined
    by your implementation.
     
    ``Teardown()`` is called once after the test is reset.
     
    The return value is ignored. Its sole purpose is to satisfy the compiler.
     
    When overwritten, it is **NOT REQUIRED** to call the base implementation ``SUPER^.Teardown()``,
    as the base implementation is empty.   
 *)
METHOD PROTECTED Teardown : BOOL
// TODO Clean up testee and test after test case finished
END_METHOD

END_FUNCTION_BLOCK

// Device/Application/Rotary/AutoRotate
FUNCTION_BLOCK AutoRotate IMPLEMENTS IAutoRotate
VAR_INPUT
	rotary: IRotary;
END_VAR
VAR_OUTPUT
END_VAR
VAR
	_enabled: BOOL;
END_VAR


{warning 'Aggiungi implementazione della proprietà'}
PROPERTY direction : STRING
GET
direction := 'LEFT';
END_GET
END_PROPERTY

{warning 'Aggiungi implementazione della proprietà'}
PROPERTY enabled : BOOL
GET
enabled := _enabled;
END_GET
SET
_enabled := enabled;
END_SET
END_PROPERTY

{warning 'Aggiungi implementazione della proprietà'}
PROPERTY speed : REAL
GET
IF enabled THEN
	speed := 20;
ELSE 
	speed := 0;
END_IF
END_GET
END_PROPERTY

END_FUNCTION_BLOCK

// Device/Application/Rotary/IAutoRotate
INTERFACE IAutoRotate

PROPERTY direction : STRING
GET
END_GET
END_PROPERTY

PROPERTY enabled : BOOL
GET
END_GET
SET
END_SET
END_PROPERTY

PROPERTY speed : REAL
GET
END_GET
END_PROPERTY

END_INTERFACE

// Device/Application/Controls/Joystyck/Joystick2
FUNCTION_BLOCK Joystick2
VAR_INPUT
END_VAR
VAR_OUTPUT
END_VAR
VAR
END_VAR

END_FUNCTION_BLOCK

// Device/Application/Controls/Joystyck/Joystick2
FUNCTION_BLOCK Joystick2
VAR_INPUT
END_VAR
VAR_OUTPUT
END_VAR
VAR
END_VAR

END_FUNCTION_BLOCK

// Device/Application/Controls/Joystyck/Joystick2
FUNCTION_BLOCK Joystick2
VAR_INPUT
END_VAR
VAR_OUTPUT
END_VAR
VAR
END_VAR

END_FUNCTION_BLOCK

// Device/Application/Controls/Joystyck/Joystick3
FUNCTION_BLOCK Joystick3
VAR_INPUT
END_VAR
VAR_OUTPUT
END_VAR
VAR
END_VAR

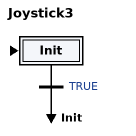
INITIAL_STEP Init:
END_STEP
TRANSITION FROM Init TO Init
    := TRUE;
END_TRANSITION

END_FUNCTION_BLOCK

// Device/Application/Controls/Joystyck/Joystick3
FUNCTION_BLOCK Joystick3
VAR_INPUT
END_VAR
VAR_OUTPUT
END_VAR
VAR
END_VAR

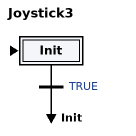
INITIAL_STEP Init:
END_STEP
TRANSITION FROM Init TO Init
    := TRUE;
END_TRANSITION

END_FUNCTION_BLOCK

// Device/Application/Controls/Joystyck/Joystick3
FUNCTION_BLOCK Joystick3
VAR_INPUT
END_VAR
VAR_OUTPUT
END_VAR
VAR
END_VAR

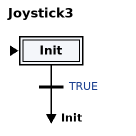
INITIAL_STEP Init:
END_STEP
TRANSITION FROM Init TO Init
    := TRUE;
END_TRANSITION

END_FUNCTION_BLOCK

// Device/Application/Visualization_1
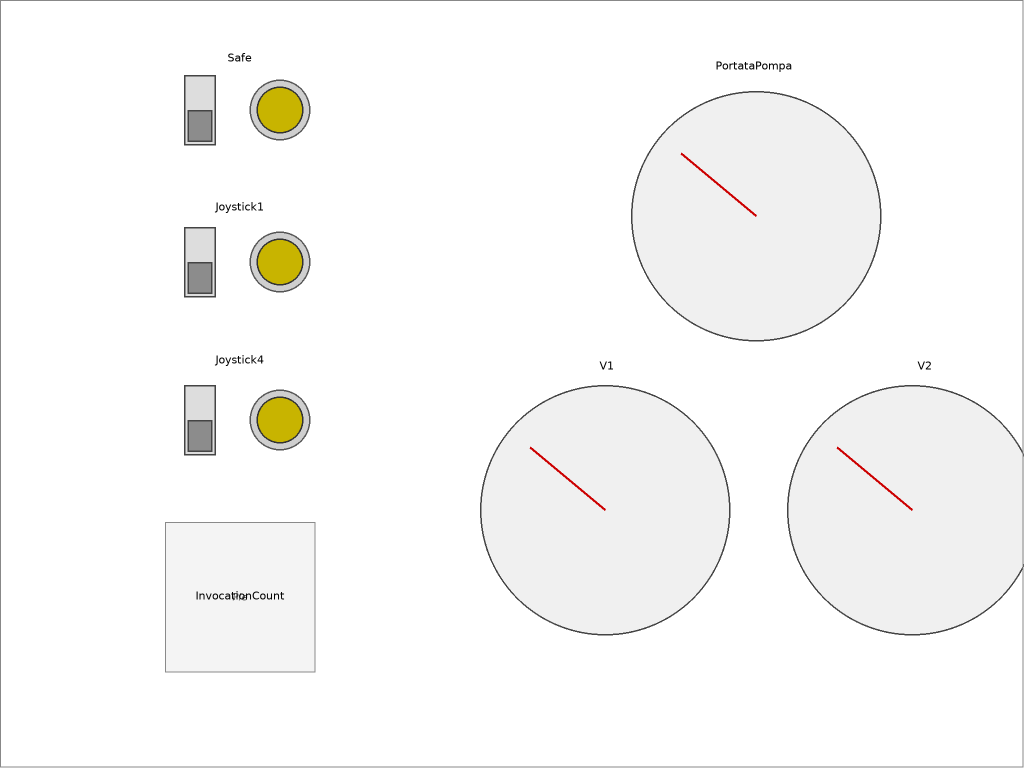
VISUALIZATION Visualization_1  // 1024x768
    DipSwitch (165,75 70x70), variable: PLC_PRG.safe, behaviour: TOGGLE, style: Switch-DipSwitch-Gray
    DipSwitch (165,385 70x70), variable: PLC_PRG.joystick.Trigger, behaviour: TOGGLE, style: Switch-DipSwitch-Gray
    Lamp1 (245,75 70x70), variable: PLC_PRG.safe, style: Lamp-Lamp1-Yellow
    DipSwitch (165,227 70x70), variable: PLC_PRG.joystick1.Trigger, behaviour: TOGGLE, style: Switch-DipSwitch-Gray
    Label (165,345 150x30), "Joystick4"
    Label (165,192 150x30), "Joystick1"
    Label (165,43 150x30), "Safe"
    Pie (165,522 150x150)
        p426801730: PLC_PRG.rotary.InvocationCount
    Label (165,581 150x30), "InvocationCount"
    Meter360 (631,91 250x250), value: PLC_PRG.pompa.portata, style: Meter-Meter360-Gray, scale format: %.1f, scale 0..100
    Meter360 (480,385 250x250), value: PLC_PRG.distributore.v1, style: Meter-Meter360-Gray, scale format: %.1f, scale 0..100
    Meter360 (787,385 250x250), value: PLC_PRG.distributore.v2, style: Meter-Meter360-Gray, scale format: %.1f, scale 0..100
    Lamp1 (245,227 70x70), variable: PLC_PRG.joystick1.Enabled, style: Lamp-Lamp1-Yellow
    Lamp1 (245,385 70x70), variable: PLC_PRG.joystick.Enabled, style: Lamp-Lamp1-Yellow
    Label (679,51 150x30), "PortataPompa"
    Label (532,351 150x30), "V1"
    Label (850,351 150x30), "V2"
END_VISUALIZATION

// Device/Application/Visualization_1
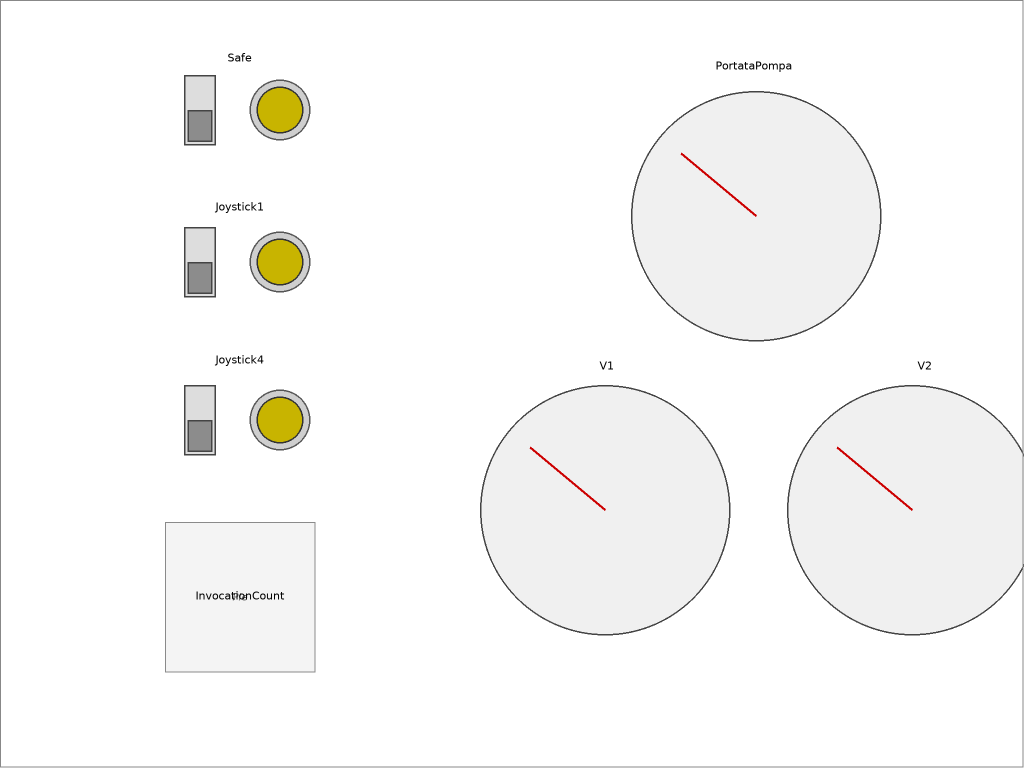
VISUALIZATION Visualization_1  // 1024x768
    DipSwitch (165,75 70x70), variable: PLC_PRG.safe, behaviour: TOGGLE, style: Switch-DipSwitch-Gray
    DipSwitch (165,385 70x70), variable: PLC_PRG.joystick.Trigger, behaviour: TOGGLE, style: Switch-DipSwitch-Gray
    Lamp1 (245,75 70x70), variable: PLC_PRG.safe, style: Lamp-Lamp1-Yellow
    DipSwitch (165,227 70x70), variable: PLC_PRG.joystick1.Trigger, behaviour: TOGGLE, style: Switch-DipSwitch-Gray
    Label (165,345 150x30), "Joystick4"
    Label (165,192 150x30), "Joystick1"
    Label (165,43 150x30), "Safe"
    Pie (165,522 150x150)
        p426801730: PLC_PRG.rotary.InvocationCount
    Label (165,581 150x30), "InvocationCount"
    Meter360 (631,91 250x250), value: PLC_PRG.pompa.portata, style: Meter-Meter360-Gray, scale format: %.1f, scale 0..100
    Meter360 (480,385 250x250), value: PLC_PRG.distributore.v1, style: Meter-Meter360-Gray, scale format: %.1f, scale 0..100
    Meter360 (787,385 250x250), value: PLC_PRG.distributore.v2, style: Meter-Meter360-Gray, scale format: %.1f, scale 0..100
    Lamp1 (245,227 70x70), variable: PLC_PRG.joystick1.Enabled, style: Lamp-Lamp1-Yellow
    Lamp1 (245,385 70x70), variable: PLC_PRG.joystick.Enabled, style: Lamp-Lamp1-Yellow
    Label (679,51 150x30), "PortataPompa"
    Label (532,351 150x30), "V1"
    Label (850,351 150x30), "V2"
END_VISUALIZATION

// Device/Application/Visualization_1
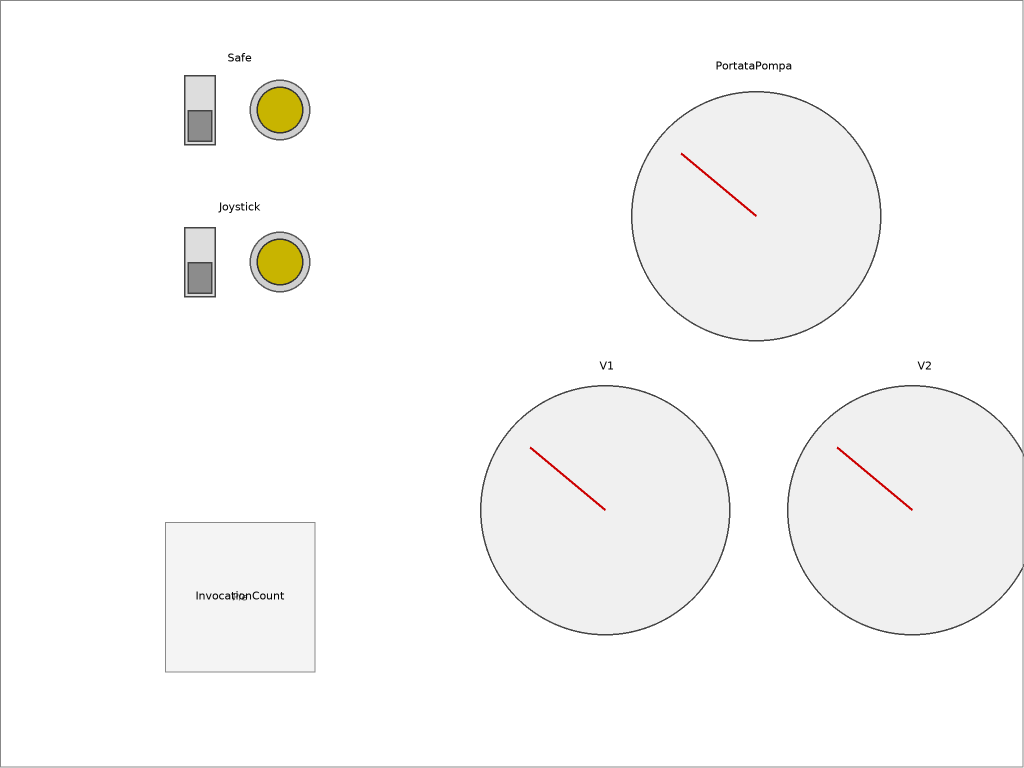
VISUALIZATION Visualization_1  // 1024x768
    DipSwitch (165,75 70x70), variable: PLC_PRG.safe, behaviour: TOGGLE, style: Switch-DipSwitch-Gray
    Lamp1 (245,75 70x70), variable: PLC_PRG.safe, style: Lamp-Lamp1-Yellow
    DipSwitch (165,227 70x70), variable: PLC_PRG.joystick._triggered, behaviour: TOGGLE, style: Switch-DipSwitch-Gray
    Label (165,192 150x30), "Joystick"
    Label (165,43 150x30), "Safe"
    Pie (165,522 150x150)
        p426801730: PLC_PRG.rotary.invocationCount
    Label (165,581 150x30), "InvocationCount"
    Meter360 (631,91 250x250), value: PLC_PRG.pump.flow, style: Meter-Meter360-Gray, scale format: %.1f, scale 0..100
    Meter360 (480,385 250x250), value: PLC_PRG.distributionValve._vActual[1], style: Meter-Meter360-Gray, scale format: %.1f, scale 0..100
    Meter360 (787,385 250x250), value: PLC_PRG.distributionValve._vActual[2], style: Meter-Meter360-Gray, scale format: %.1f, scale 0..100
    Lamp1 (245,227 70x70), variable: PLC_PRG.joystick._triggered, style: Lamp-Lamp1-Yellow
    Label (679,51 150x30), "PortataPompa"
    Label (532,351 150x30), "V1"
    Label (850,351 150x30), "V2"
END_VISUALIZATION
